PROGRAM MAIN
VAR
	
	// Declare FB_IotCommunicator
	fbIot : FB_IotCommunicator := (sHostName := 'iot.beckhoff.us',
									nPort := 1883,
									sMainTopic := 'Test',
									sDeviceName := 'Automated Building',
									sDeviceIcon := 'House');
	
	// Timer to send data only once per second
	timer : TON;
	
	
	

END_VAR

// .Execute() has to be called cyclically
fbIot.Execute(TRUE);

// Start timer when fbIot is connected
IF fbIot.bConnected THEN
	timer(IN := TRUE, PT := T#500MS);
END_IF


// Send data, if timer is expired
IF timer.Q THEN
	timer(IN := FALSE);
	fbIot.SendData(ADR(House.stFloorOne), SIZEOF(House.stFloorOne));
END_IF



Lighting(); 
Constants();
Room_One();

METHOD Lighting 
VAR_INPUT
END_VAR
IF fbIot.fbCommand.bAvailable THEN
	// Receive data for first level struct

	IF fbIot.fbCommand.sVarName = 'stLights.stLighting.bLight' THEN
		fbIot.fbCommand.GetValue(ADR(House.stFloorOne.stLights.stLighting.bLight), SIZEOF(House.stFloorOne.stLights.stLighting.bLight), E_IotCommunicatorDatatype.type_BOOL);
	ELSIF fbIot.fbCommand.sVarName = 'stLights.stLighting.nLight' THEN
		fbIot.fbCommand.GetValue(ADR(House.stFloorOne.stLights.stLighting.nLight), SIZEOF(House.stFloorOne.stLights.stLighting.nLight), E_IotCommunicatorDatatype.type_INT);
	ELSIF fbIot.fbCommand.sVarName = 'stLights.stLighting.sMode' THEN
		fbIot.fbCommand.GetValue(ADR(House.stFloorOne.stLights.stLighting.sMode), SIZEOF(House.stFloorOne.stLights.stLighting.sMode), E_IotCommunicatorDatatype.type_STRING);
	END_IF
	fbIot.SendData(ADR(House.stFloorOne), SIZEOF(House.stFloorOne));
	fbIot.fbCommand.Remove();
END_IF

//Lighting Sample 2
House.stFloorOne.stLights.stLighting.aModes[0]:='Automatic';
House.stFloorOne.stLights.stLighting.aModes[1]:='Manual';
END_METHOD

METHOD Room_One 
VAR_INPUT
END_VAR
IF fbIot.fbCommand.bAvailable THEN
	// Receive data for first level struct

	IF fbIot.fbCommand.sVarName = 'stRoomOne.Projector' THEN
		fbIot.fbCommand.GetValue(ADR(House.stFloorOne.stRoomOne.Projector), SIZEOF(House.stFloorOne.stRoomOne.Projector), E_IotCommunicatorDatatype.type_BOOL);
	END_IF
	
	IF fbIot.fbCommand.sVarName = 'stRoomOne.ConTemp' THEN
		fbIot.fbCommand.GetValue(ADR(House.stFloorOne.stRoomOne.ConTemp), SIZEOF(House.stFloorOne.stRoomOne.ConTemp), E_IotCommunicatorDatatype.type_LREAL);
	END_IF
	
	fbIot.SendData(ADR(House.stFloorOne), SIZEOF(House.stFloorOne));
	fbIot.fbCommand.Remove();
END_IF
END_METHOD

END_PROGRAM

(* stored: Version 1.1.0.1, ProductVersion 3.1.4024.12
   POU MAIN: Id {44b9cdcb-0c7c-4675-bb09-0840c2c77ec3}, SpecialFunc None
   Method Lighting: Id {f962bd32-f177-4d94-a573-5170c5142db5}
   Method Room_One: Id {7de3a368-7e3a-4ce6-9c00-29fa850e5b79} *)
